PROGRAM schudmachine
VAR
	State : schudmachineToestand;
	schudmachineReady : BOOL := FALSE;
	schudMachineBezig : BOOL := FALSE;
	deurDicht : BOOL := FALSE;
	stopSchudden : BOOL := FALSE;
	blikGevonden : BOOL := FALSE;
	geenBlikGevonden : BOOL;
	//fBlikKlemmen : BlikKlemmen;
	
	timerSchudMachine : TON;
	klemTimer : TON;
	blikGeklemd: BOOL;
	geenBlik: BOOL;
END_VAR

CASE State OF
	schudMachineToestand.startup:
		// Simulate startup
		timerSchudMachine(IN:=TRUE,PT:=T#5S);
		IF timerSchudMachine.Q THEN
			State := schudMachineToestand.automode;
			timerSchudMachine(IN:=FALSE);
		END_IF
		
	schudMachineToestand.automode:
		// CODE
		schudmachineReady := TRUE;
		schudmachineBezig := FALSE;
		IF deurDicht THEN
			State := schudmachineToestand.blikKlemmen;
		END_IF

	schudMachineToestand.blikKlemmen:
		// CODE
		schudmachineReady := FALSE;
		schudmachineBezig := TRUE;
		
		// clamping procedure
		klemTimer(IN:=TRUE, PT:= T#10S);
		IF klemTimer.ET = T#7S THEN // simulate finding the can with the clamp
			blikGevonden := TRUE;
			klemTimer(IN:=FALSE);
		ELSIF klemTimer.Q THEN // if no can is found
			geenBlik := TRUE;
		END_IF
		
		// checks to change state
		IF blikGevonden THEN
			State := schudmachineToestand.blikSchudden;
		ELSIF stopSchudden THEN
			State := schudmachineToestand.automode;
			deurDicht := FALSE;
		ELSIF geenBlik THEN
			State := schudmachineToestand.automode;
			deurDicht := FALSE;
		END_IF
		
	schudMachineToestand.blikSchudden:
		// CODE
		timerSchudMachine(IN:=TRUE, PT:= T#1M);
		IF timerSchudMachine.Q THEN
			State := schudmachineToestand.automode;
			deurDicht := FALSE;
		ELSIF stopSchudden THEN
			State := schudmachineToestand.automode;
			deurDicht := FALSE;
		END_IF
	
END_CASE

END_PROGRAM

(* stored: Version 1.1.0.1, ProductVersion 3.1.4024.15
   POU schudmachine: Id {0b29f726-389e-47ee-8ec4-583a70285669}, SpecialFunc None *)
